// This is actaully just ANY without pointer
TYPE ListType :
STRUCT
	size		: DINT;
	typeClass	: __SYSTEM.TYPE_CLASS;
	typeName	: T_MaxString;
END_STRUCT
END_TYPE

(* stored: Version 1.1.0.1, ProductVersion 3.1.4024.12
   DUT ListType: Id {6a1bef6b-213c-4cce-a9c0-8b161d18637a} *)
